Fanuc KAREL source: kt00412.KL

-- PROVISIONAL review KL for V770-1; original PC SHA256 35bc8027eb9a8b277f7d7128b2dbce1f16d63e4292240c5d34d2f4541fc9801d
-- Incomplete behavior may be omitted. Consult companion uncertainty JSON. Do not deploy.
PROGRAM KT00412
%NOLOCKGROUP
VAR
  R2 : REAL
  OUT : BOOLEAN
-- UNRESOLVED_DECL Y1 type=002018
BEGIN
  -- UNRESOLVED_PC offsets 5-19; opcodes 2E,22,9D,33,B2
  -- UNRESOLVED_PC offsets 24-35; opcodes 2E,23
  -- UNRESOLVED_PC offsets 40-65; opcodes 22,9D,33,B1,21,29,64,29,71,23
  -- UNRESOLVED_PC offsets 70-74; opcodes 7F
END KT00412
